// Brief: Master Arm Test
FUNCTION_BLOCK PUBLIC FB_StateCtrlTest EXTENDS FB_MasterArmCtrlBase
VAR_INPUT
END_VAR
VAR_OUTPUT
END_VAR
VAR
	// ################ variables for single DH  joint test ##################
	m_freqTestFlag :BOOL:=FALSE;
	m_initJntPos :Vec7d;
	m_jntMotionFreq :Vec7d :=[0.2, 0.2, 0.1, 4(0.1)];
	m_jntMotionRange :Vec7d :=[pi/6, pi/6, 0.1, 4(pi/6)];
	m_testJntIdx :INT :=1;
	
	m_stepTestFlag :BOOL :=FALSE;
	m_jntStep : LREAL := 5*g_deg2Rad;
	
END_VAR

METHOD PROTECTED calcCmdJntPos : BOOL
VAR_IN_OUT CONSTANT
	i_slaveIdx :INT;
	i_shoulderPose :ST_Frame;
	i_masterArm :FB_MasterArm;
	i_slaveStatus :ST_SlaveStatus;
END_VAR

VAR 
	i:INT :=0;
	errThres :LREAL;
	m_masterGripAngle: INT;
END_VAR
// Just for joint controller test
IF m_testJntIdx >=1 AND m_testJntIdx <=7 THEN
	IF m_freqTestFlag THEN 
		m_cmdJntPos[m_testJntIdx]:=m_initJntPos[m_testJntIdx]+m_jntMotionRange[m_testJntIdx]/2
										+0.5*m_jntMotionRange[m_testJntIdx]*SIN(2*pi*m_jntMotionFreq[m_testJntIdx]*m_timePeriod-pi/2);
		m_cmdJntVel[m_testJntIdx]:=0.5*m_jntMotionRange[m_testJntIdx]*2*pi*m_jntMotionFreq[m_testJntIdx]*COS(2*pi*m_jntMotionFreq[m_testJntIdx]*m_timePeriod-pi/2);
	ELSIF m_stepTestFlag THEN
		m_cmdJntPos[m_testJntIdx]:=m_initJntPos[m_testJntIdx]+m_jntStep;
		m_cmdJntVel[m_testJntIdx]:=0;
	ELSE
		m_timePeriod:=0;
	END_IF
	
END_IF


FOR i:=1 TO 3 DO 
		errThres :=5*g_deg2rad;
	IF ABS(m_cmdJntPos[i]-i_masterArm.curJntPos[i])>errThres THEN
		m_isFinished:=TRUE;
	END_IF
	
END_FOR
END_METHOD

METHOD PUBLIC init : BOOL
VAR_IN_OUT CONSTANT
	i_masterArm	:FB_MasterArm;
END_VAR
VAR_IN_OUT 
	r_masterArmCtrlCmd :ST_ArmCtrlCmds;
END_VAR
// check if to hold the command joint position unchanged
m_holdLastCmds := checkToHoldLastCmds(i_masterArm);

// init
SUPER^.Init(i_masterArm,r_masterArmCtrlCmd);

m_initJntPos := i_masterArm.curJntPos;
END_METHOD

END_FUNCTION_BLOCK

(* stored: Version 1.1.0.1, ProductVersion 3.1.4024.12
   POU FB_StateCtrlTest: Id {0c47bb14-eaef-4d00-89db-6153e5307754}, SpecialFunc None
   Method calcCmdJntPos: Id {010d1f8e-611a-45d6-a3e6-a98e946007a3}
   Method init: Id {577e5bac-bcb1-4cc3-b600-c297bc6f4cb5} *)
